{attribute addProperty BoxType "KL3001"}
{attribute addProperty Id "Channel_1Channel_B0A8062F00"}
{attribute addProperty CRC "2809087995"}
{attribute addProperty SizeInBites "0"}
{attribute addProperty SizeInBytes "0"}
TYPE KL3001_A76F47FB :
STRUCT
	{attribute addProperty Name "Channel_1"}
	Channel_1 : Channel_B0A8062F;
END_STRUCT
END_TYPE

(* stored: Version 1.2.0.0, ProductVersion 3.1.4024.9
   DUT KL3001_A76F47FB: Id {4a6233b9-a5bb-497b-b82c-db1e96b1d6e5} *)
